// TIA Portal V15.1 export
// export: Created 2020-06-12T07:35:44.5849609Z, ExportSetting None, DisplayName Totally Integrated Automation Portal, DisplayVersion V15.1, DisplayName TIA Portal Openness, DisplayVersion V15.1, DisplayName STEP 7 Professional, DisplayVersion V15.1, DisplayName STEP 7 Safety, DisplayVersion V15.1, DisplayName WinCC Advanced, DisplayVersion V15.1
FUNCTION "HMI_MSG" : Void   // FC130, FBD
{ S7_Optimized_Access := 'TRUE' }
// stored: SetENOAutomatically False
   VAR_TEMP
      _ht_wt : Real;
   END_VAR
BEGIN

REGION Network 1: Message: Emergency not OK
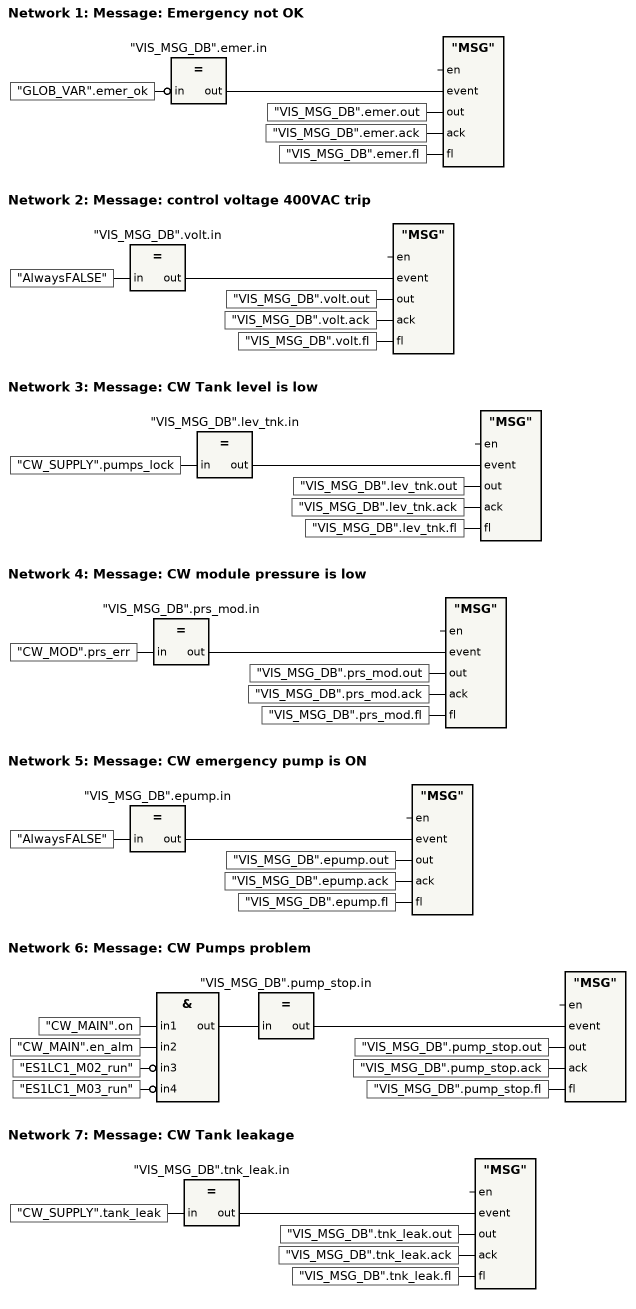
   "VIS_MSG_DB".emer.in := NOT "GLOB_VAR".emer_ok;
   "MSG"(event := NOT "GLOB_VAR".emer_ok,
         out := "VIS_MSG_DB".emer.out,
         ack := "VIS_MSG_DB".emer.ack,
         fl := "VIS_MSG_DB".emer.fl);
END_REGION

REGION Network 2: Message: control voltage 400VAC trip
   // "ES1GM01_volt_trp"
   "VIS_MSG_DB".volt.in := "AlwaysFALSE";
   "MSG"(event := "AlwaysFALSE",
         out := "VIS_MSG_DB".volt.out,
         ack := "VIS_MSG_DB".volt.ack,
         fl := "VIS_MSG_DB".volt.fl);
END_REGION

REGION Network 3: Message: CW Tank level is low
   "VIS_MSG_DB".lev_tnk.in := "CW_SUPPLY".pumps_lock;
   "MSG"(event := "CW_SUPPLY".pumps_lock,
         out := "VIS_MSG_DB".lev_tnk.out,
         ack := "VIS_MSG_DB".lev_tnk.ack,
         fl := "VIS_MSG_DB".lev_tnk.fl);
END_REGION

REGION Network 4: Message: CW module pressure is low
   "VIS_MSG_DB".prs_mod.in := "CW_MOD".prs_err;
   "MSG"(event := "CW_MOD".prs_err,
         out := "VIS_MSG_DB".prs_mod.out,
         ack := "VIS_MSG_DB".prs_mod.ack,
         fl := "VIS_MSG_DB".prs_mod.fl);
END_REGION

REGION Network 5: Message: CW emergency pump is ON
   // "stat_ES1LC1".M01.auto_on
   "VIS_MSG_DB".epump.in := "AlwaysFALSE";
   "MSG"(event := "AlwaysFALSE",
         out := "VIS_MSG_DB".epump.out,
         ack := "VIS_MSG_DB".epump.ack,
         fl := "VIS_MSG_DB".epump.fl);
END_REGION

REGION Network 6: Message: CW Pumps problem
   "VIS_MSG_DB".pump_stop.in := "CW_MAIN".on AND "CW_MAIN".en_alm AND NOT "ES1LC1_M02_run" AND NOT "ES1LC1_M03_run";
   "MSG"(event := "VIS_MSG_DB".pump_stop.in,
         out := "VIS_MSG_DB".pump_stop.out,
         ack := "VIS_MSG_DB".pump_stop.ack,
         fl := "VIS_MSG_DB".pump_stop.fl);
END_REGION

REGION Network 7: Message: CW Tank leakage
   "VIS_MSG_DB".tnk_leak.in := "CW_SUPPLY".tank_leak;
   "MSG"(event := "CW_SUPPLY".tank_leak,
         out := "VIS_MSG_DB".tnk_leak.out,
         ack := "VIS_MSG_DB".tnk_leak.ack,
         fl := "VIS_MSG_DB".tnk_leak.fl);
END_REGION

REGION Network 8: Message: CW Emergency water is open
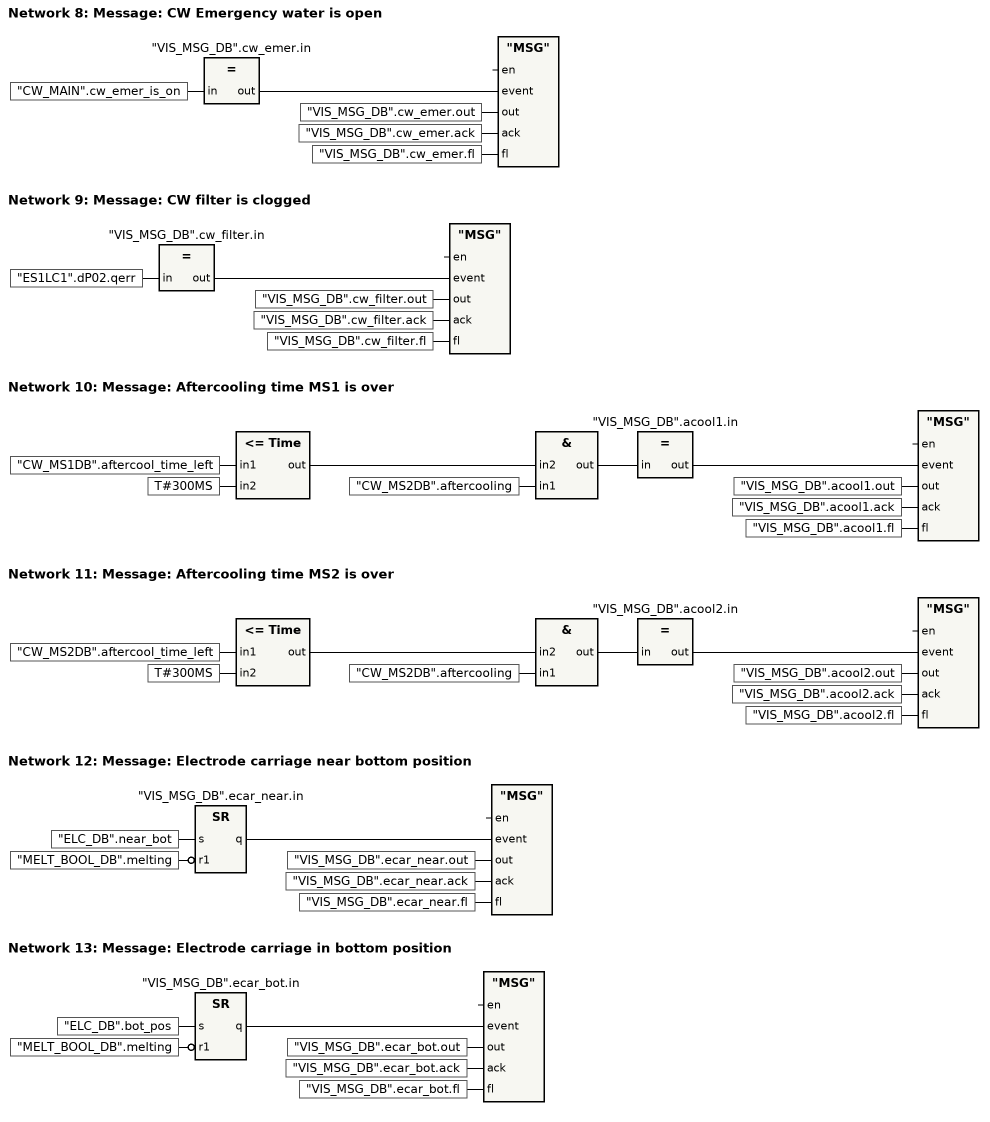
   "VIS_MSG_DB".cw_emer.in := "CW_MAIN".cw_emer_is_on;
   "MSG"(event := "CW_MAIN".cw_emer_is_on,
         out := "VIS_MSG_DB".cw_emer.out,
         ack := "VIS_MSG_DB".cw_emer.ack,
         fl := "VIS_MSG_DB".cw_emer.fl);
END_REGION

REGION Network 9: Message: CW filter is clogged
   "VIS_MSG_DB".cw_filter.in := "ES1LC1".dP02.qerr;
   "MSG"(event := "ES1LC1".dP02.qerr,
         out := "VIS_MSG_DB".cw_filter.out,
         ack := "VIS_MSG_DB".cw_filter.ack,
         fl := "VIS_MSG_DB".cw_filter.fl);
END_REGION

REGION Network 10: Message: Aftercooling time MS1 is over
   "VIS_MSG_DB".acool1.in := ("CW_MS1DB".aftercool_time_left <= T#300MS) AND "CW_MS2DB".aftercooling;
   "MSG"(event := "VIS_MSG_DB".acool1.in,
         out := "VIS_MSG_DB".acool1.out,
         ack := "VIS_MSG_DB".acool1.ack,
         fl := "VIS_MSG_DB".acool1.fl);
END_REGION

REGION Network 11: Message: Aftercooling time MS2 is over
   "VIS_MSG_DB".acool2.in := ("CW_MS2DB".aftercool_time_left <= T#300MS) AND "CW_MS2DB".aftercooling;
   "MSG"(event := "VIS_MSG_DB".acool2.in,
         out := "VIS_MSG_DB".acool2.out,
         ack := "VIS_MSG_DB".acool2.ack,
         fl := "VIS_MSG_DB".acool2.fl);
END_REGION

REGION Network 12: Message: Electrode carriage near bottom position
   IF "ELC_DB".near_bot THEN
       "VIS_MSG_DB".ecar_near.in := TRUE;   // SR flip-flop
   END_IF;
   IF NOT "MELT_BOOL_DB".melting THEN "VIS_MSG_DB".ecar_near.in := FALSE; END_IF;
   "MSG"(event := "VIS_MSG_DB".ecar_near.in,
         out := "VIS_MSG_DB".ecar_near.out,
         ack := "VIS_MSG_DB".ecar_near.ack,
         fl := "VIS_MSG_DB".ecar_near.fl);
END_REGION

REGION Network 13: Message: Electrode carriage in bottom position
   IF "ELC_DB".bot_pos THEN
       "VIS_MSG_DB".ecar_bot.in := TRUE;   // SR flip-flop
   END_IF;
   IF NOT "MELT_BOOL_DB".melting THEN "VIS_MSG_DB".ecar_bot.in := FALSE; END_IF;
   "MSG"(event := "VIS_MSG_DB".ecar_bot.in,
         out := "VIS_MSG_DB".ecar_bot.out,
         ack := "VIS_MSG_DB".ecar_bot.ack,
         fl := "VIS_MSG_DB".ecar_bot.fl);
END_REGION

REGION Network 14: Message: Hottopping starts in 1 minute
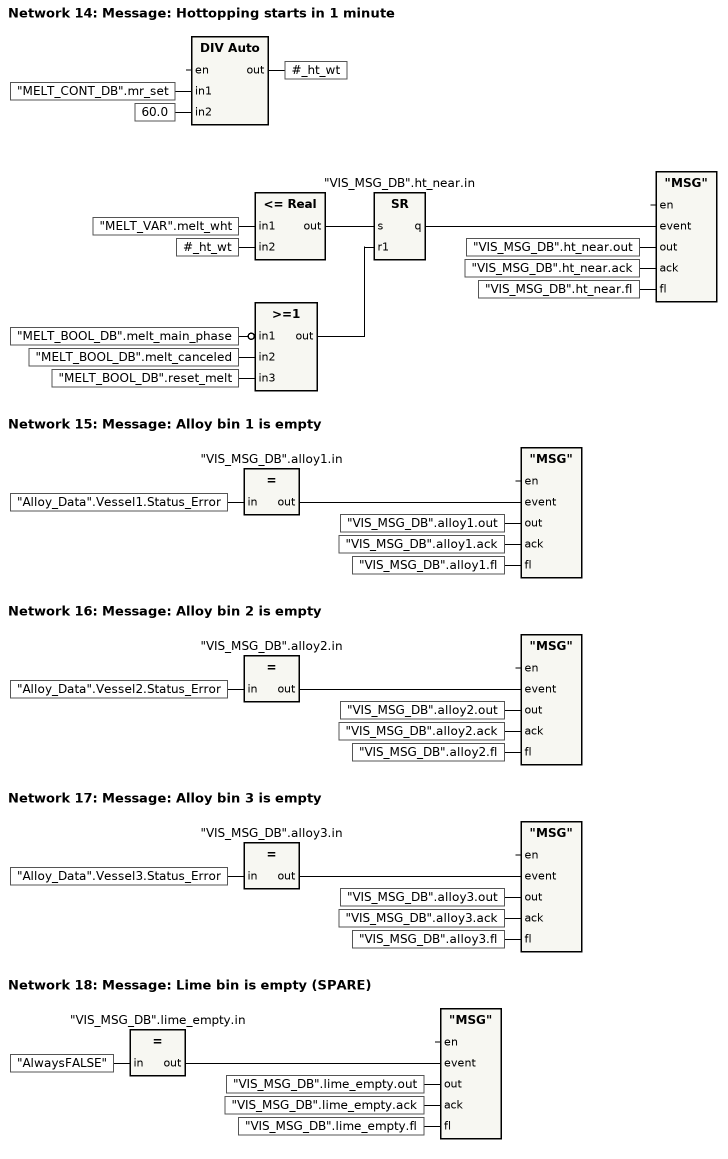
   #_ht_wt := "MELT_CONT_DB".mr_set / 60.0;
   IF "MELT_VAR".melt_wht <= #_ht_wt THEN
       "VIS_MSG_DB".ht_near.in := TRUE;   // SR flip-flop
   END_IF;
   IF NOT "MELT_BOOL_DB".melt_main_phase OR "MELT_BOOL_DB".melt_canceled OR "MELT_BOOL_DB".reset_melt THEN
       "VIS_MSG_DB".ht_near.in := FALSE;
   END_IF;
   "MSG"(event := "VIS_MSG_DB".ht_near.in,
         out := "VIS_MSG_DB".ht_near.out,
         ack := "VIS_MSG_DB".ht_near.ack,
         fl := "VIS_MSG_DB".ht_near.fl);
END_REGION

REGION Network 15: Message: Alloy bin 1 is empty
   "VIS_MSG_DB".alloy1.in := "Alloy_Data".Vessel1.Status_Error;
   "MSG"(event := "Alloy_Data".Vessel1.Status_Error,
         out := "VIS_MSG_DB".alloy1.out,
         ack := "VIS_MSG_DB".alloy1.ack,
         fl := "VIS_MSG_DB".alloy1.fl);
END_REGION

REGION Network 16: Message: Alloy bin 2 is empty
   "VIS_MSG_DB".alloy2.in := "Alloy_Data".Vessel2.Status_Error;
   "MSG"(event := "Alloy_Data".Vessel2.Status_Error,
         out := "VIS_MSG_DB".alloy2.out,
         ack := "VIS_MSG_DB".alloy2.ack,
         fl := "VIS_MSG_DB".alloy2.fl);
END_REGION

REGION Network 17: Message: Alloy bin 3 is empty
   "VIS_MSG_DB".alloy3.in := "Alloy_Data".Vessel3.Status_Error;
   "MSG"(event := "Alloy_Data".Vessel3.Status_Error,
         out := "VIS_MSG_DB".alloy3.out,
         ack := "VIS_MSG_DB".alloy3.ack,
         fl := "VIS_MSG_DB".alloy3.fl);
END_REGION

REGION Network 18: Message: Lime bin is empty (SPARE)
   "VIS_MSG_DB".lime_empty.in := "AlwaysFALSE";
   "MSG"(event := "AlwaysFALSE",
         out := "VIS_MSG_DB".lime_empty.out,
         ack := "VIS_MSG_DB".lime_empty.ack,
         fl := "VIS_MSG_DB".lime_empty.fl);
END_REGION
END_FUNCTION
